(* IEC 61131-3 sources: programs/VI-54/VI-54_20171205/VI-54_20171205/Stations/PLC_VI54/VI-54_171014/Class/SpeedInput, 1 file *)

(* ---- SpeedInput.st ---- *)
(*!
<Class
	Name               = "SpeedInput"
	Revision           = "0.0"
	RealtimeTask       = "false"
	CyclicTask         = "false"
	BackgroundTask     = "false"
	Sigmatek           = "false"
	OSInterface        = "false"
	HighPriority       = "false"
	Automatic          = "false"
	UpdateMode         = "Prescan"
	SharedCommandTable = "true"
	Objectsize         = "(480,480)">
	<Channels>
		<Server Name="__________" Visualized="false" Initialize="false" WriteProtected="true" Retentive="false"/>
		<Server Name="ActInfeedSpeed" Visualized="true" Initialize="false" WriteProtected="true" Retentive="false"/>
		<Server Name="ClassSvr" Visualized="false" Initialize="false" WriteProtected="true" Retentive="false"/>
		<Server Name="MaxAccDec" Visualized="true" Initialize="true" WriteProtected="false" Retentive="File" Comment="Maximal acceleration at 100%"/>
		<Server Name="MaxAnalogInput" Visualized="true" Initialize="true" WriteProtected="false" Retentive="File"/>
		<Server Name="MaxSpeed" Visualized="true" Initialize="true" WriteProtected="false" Retentive="File" Comment="Maximal velocity at 100%"/>
		<Server Name="PercentageOverride" Visualized="true" Initialize="false" WriteProtected="true" Retentive="false"/>
		<Server Name="PulsenPerMM" Visualized="true" Initialize="true" WriteProtected="false" Retentive="File" Comment="How many pulses do we get for 1 mm&#13;&#10;"/>
		<Client Name="iAnlogSpeed" Required="false" Internal="false"/>
		<Client Name="iEncoderPos" Required="false" Internal="false"/>
		<Client Name="Standard1" Required="true" Internal="true"/>
	</Channels>
	<Network Name="SpeedInput">
		<!-- List of Components in this network -->
		<Components>
			<Object
				Name           = "Standard1"
				Class          = "Standard"
				Position       = "(210,480)"
				Visualized     = "false"
				BackgroundTime = "1000 ms">
				<Channels>
					<Server Name="ClassSvr"/>
				</Channels>
			</Object>
		</Components>
		<Comments>
		</Comments>
		<!-- List of Connections in this network -->
		<Connections>
			<Connection Source="this.Standard1" Destination="Standard1.ClassSvr"/>
		</Connections>
		<!-- Headerfiles -->
		<Options>
		</Options>
	</Network>
</Class>
*)
SpeedInput : CLASS
	TYPE
	  eInput :  //! <Type Public="true" Name="eInput"/>
	  (
	    eAnalog,
	    eEncoder
	  )$UDINT;
	END_TYPE
  //Servers:
	ClassSvr 	: SvrChCmd_DINT;
	ActInfeedSpeed 	: SvrCh_DINT;
	PercentageOverride 	: SvrCh_DINT;
	__________ 	: SvrCh_DINT;
	MaxSpeed 	: SvrCh_DINT;
	MaxAccDec 	: SvrCh_DINT;
	MaxAnalogInput 	: SvrCh_DINT;
	PulsenPerMM 	: SvrCh_DINT;
  //Clients:
	iAnlogSpeed 	: CltCh_DINT;
	Standard1 	: CltChCmd_Standard;
	iEncoderPos 	: CltCh_DINT;
  //Variables:
		MaxPackageSpeed 	: DINT;
		MaxPackageAccDec 	: DINT;
		CalcSpeed 	: REAL;
		CalcSpeedIntUnits 	: DINT;
		OldEncoderPuls 	: DINT;
  //Functions:

	FUNCTION VIRTUAL GLOBAL ReadMaxSpeed
		VAR_OUTPUT
			Speed 	: DINT;
		END_VAR;

	FUNCTION VIRTUAL GLOBAL ReadPercentage
		VAR_OUTPUT
			Percentage 	: DINT;
		END_VAR;

	FUNCTION VIRTUAL GLOBAL ReadMaxAcceleration
		VAR_OUTPUT
			Acceleration 	: DINT;
		END_VAR;

	FUNCTION GLOBAL EncoderInput;

	FUNCTION GLOBAL AnalogInput;

	FUNCTION GLOBAL ResetEncoderInput;

	FUNCTION GLOBAL MyRtTask
		VAR_INPUT
			InputSetting 	: eInput;
		END_VAR;
  //Tables:
	FUNCTION @STD
		VAR_OUTPUT
			ret_code	: CONFSTATES;
		END_VAR;
	FUNCTION GLOBAL TAB @CT_;
END_CLASS;

#pragma using Standard

FUNCTION GLOBAL SpeedInput::MyRtTask
	VAR_INPUT
		InputSetting 	: eInput;
	END_VAR

  if InputSetting = eAnalog then
    AnalogInput();
  elsif InputSetting = eEncoder then
    EncoderInput();
  end_if;

  // Calculate Max speed and Max acceleration
  MaxPackageSpeed  := to_dint(to_real MaxSpeed ToMMperSec);
  MaxPackageAccDec := to_dint(to_real MaxAccDec ToMMperSec2);

END_FUNCTION

FUNCTION VIRTUAL GLOBAL SpeedInput::ReadMaxSpeed
	VAR_OUTPUT
		Speed 	: DINT;
	END_VAR

  Speed := MaxPackageSpeed;

END_FUNCTION

FUNCTION VIRTUAL GLOBAL SpeedInput::ReadPercentage
	VAR_OUTPUT
		Percentage 	: DINT;
	END_VAR

  Percentage := PercentageOverride;

END_FUNCTION

FUNCTION VIRTUAL GLOBAL SpeedInput::ReadMaxAcceleration
	VAR_OUTPUT
		Acceleration 	: DINT;
	END_VAR

  Acceleration := MaxPackageAccDec;

END_FUNCTION

FUNCTION GLOBAL SpeedInput::AnalogInput

  iAnlogSpeed := iAnlogSpeed.Read();

  // Percentage override
  if iAnlogSpeed > 10 then
    PercentageOverride := to_dint(to_real iAnlogSpeed / 10.0);
  else
    PercentageOverride := 0;
  end_if;

  ActInfeedSpeed := to_dint(to_real MaxSpeed * (to_real iAnlogSpeed / MaxAnalogInput));

END_FUNCTION

FUNCTION GLOBAL SpeedInput::EncoderInput

  iEncoderPos := iEncoderPos.Read();
  // We divide it by 4 because our cyclic time is 4ms (Calcspeed is in m/min in xxx.x)
  CalcSpeed         := (((to_real (iEncoderPos- OldEncoderPuls) / to_Real PulsenPerMM) / 4.0) * 600.0);
  CalcSpeedIntUnits := to_dint(to_real CalcSpeed ToMMperSec);
  OldEncoderPuls    := iEncoderPos;

  PercentageOverride := to_dint((to_Real CalcSpeedIntUnits * 1000.0) / to_real MaxPackageSpeed);

END_FUNCTION

FUNCTION GLOBAL SpeedInput::ResetEncoderInput

  // Reset the encoder counter
  iEncoderPos.Write(input:= 0);

END_FUNCTION
